# EPICS substitutions: iocs/micosIOC/iocBoot/iocMicos/MoCo.substitutions
file "$(MOTOR)/db/motor.db"
{
pattern
{P,         N,      M,      DTYP,        C,  S,  DESC,          EGU,      DIR,  VELO,  VBAS,  ACCL,  BDST,  BVEL,  BACC,  MRES,  PREC,  DHLM,  DLLM,  INIT}
{micos:,    1,  "m$(N)",  "Micos MoCo",  0,  0,  "motor $(N)",  degrees,  Pos,  1,     .1,    .2,    0,     1,     .2,    0.01,  5,     100,   -100,  ""}
{micos:,    2,  "m$(N)",  "Micos MoCo",  0,  1,  "motor $(N)",  degrees,  Pos,  1,     .1,    .2,    0,     1,     .2,    0.01,  5,     100,   -100,  ""}
}
